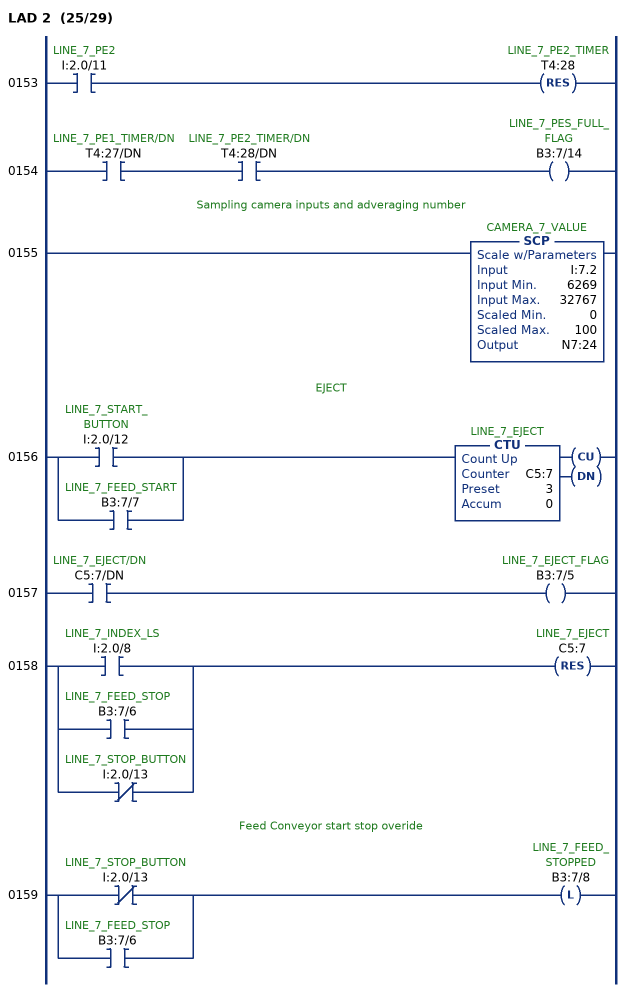
% Rung: 153 %  % edit flag set %
SOR XIC I:2.0/11 RES T4:28 EOR
%   I:2.0/11  LINE_7_PE2 %
%   T4:28  LINE_7_PE2_TIMER %
% Rung: 154 %  % edit flag set %
SOR XIC T4:27/DN XIC T4:28/DN OTE B3:7/14 EOR
%   T4:27  LINE_7_PE1_TIMER %
%   T4:28  LINE_7_PE2_TIMER %
%   B3:7/14  LINE_7_PES_FULL_FLAG %
% Rung: 155 %  % edit flag set %
% Sampling camera inputs and adveraging number %
SOR SCP I:7.2 6269 32767 0 100 N7:24 EOR
%   N7:24  CAMERA_7_VALUE %
% Rung: 156 %  % edit flag set %
% EJECT %
SOR BST XIC I:2.0/12 NXB XIC B3:7/7 BND CTU C5:7 3 0 EOR
%   I:2.0/12  LINE_7_START_BUTTON %
%   B3:7/7  LINE_7_FEED_START %
%   C5:7  LINE_7_EJECT %
% Rung: 157 %  % edit flag set %
SOR XIC C5:7/DN OTE B3:7/5 EOR
%   C5:7  LINE_7_EJECT %
%   B3:7/5  LINE_7_EJECT_FLAG %
% Rung: 158 %  % edit flag set %
SOR BST XIC I:2.0/8 NXB BST XIC B3:7/6 NXB XIO I:2.0/13 BND BND RES C5:7 EOR
%   I:2.0/8  LINE_7_INDEX_LS %
%   B3:7/6  LINE_7_FEED_STOP %
%   I:2.0/13  LINE_7_STOP_BUTTON %
%   C5:7  LINE_7_EJECT %
% Rung: 159 %  % edit flag set %
% Feed Conveyor start stop overide %
SOR BST XIO I:2.0/13 NXB XIC B3:7/6 BND OTL B3:7/8 EOR
%   I:2.0/13  LINE_7_STOP_BUTTON %
%   B3:7/6  LINE_7_FEED_STOP %
%   B3:7/8  LINE_7_FEED_STOPPED %

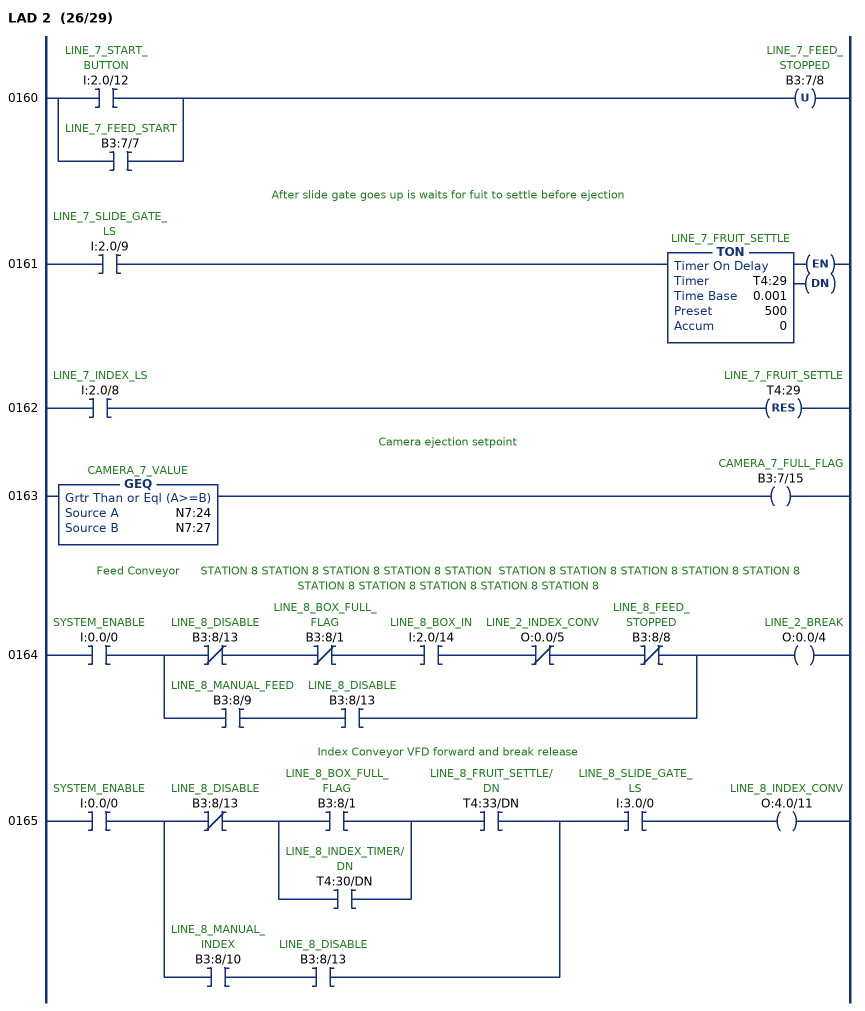
% Rung: 160 %  % edit flag set %
SOR BST XIC I:2.0/12 NXB XIC B3:7/7 BND OTU B3:7/8 EOR
%   I:2.0/12  LINE_7_START_BUTTON %
%   B3:7/7  LINE_7_FEED_START %
%   B3:7/8  LINE_7_FEED_STOPPED %
% Rung: 161 %  % edit flag set %
% After slide gate goes up is waits for fuit to settle before ejection %
SOR XIC I:2.0/9 TON T4:29 0.001 500 0 EOR
%   I:2.0/9  LINE_7_SLIDE_GATE_LS %
%   T4:29  LINE_7_FRUIT_SETTLE %
% Rung: 162 %  % edit flag set %
SOR XIC I:2.0/8 RES T4:29 EOR
%   I:2.0/8  LINE_7_INDEX_LS %
%   T4:29  LINE_7_FRUIT_SETTLE %
% Rung: 163 %  % edit flag set %
% Camera ejection setpoint %
SOR GEQ N7:24 N7:27 OTE B3:7/15 EOR
%   N7:24  CAMERA_7_VALUE %
%   N7:27  CAMERA_7_EJECT %
%   B3:7/15  CAMERA_7_FULL_FLAG %
% Rung: 164 %  % edit flag set %
% Feed Conveyor      STATION 8 STATION 8 STATION 8 STATION 8 STATION  STATION 8 STATION 8 STATION 8 STATION 8 STATION 8 STATION 8 STATION 8 STATION 8 STATION 8 STATION 8 %
SOR XIC I:0.0/0 BST XIO B3:8/13 XIO B3:8/1 XIC I:2.0/14 XIO O:0.0/5 XIO B3:8/8 NXB XIC B3:8/9 XIC B3:8/13 BND OTE O:0.0/4 EOR
%   I:0.0/0  SYSTEM_ENABLE %
%   B3:8/13  LINE_8_DISABLE %
%   B3:8/1  LINE_8_BOX_FULL_FLAG %
%   I:2.0/14  LINE_8_BOX_IN %
%   O:0.0/5  LINE_2_INDEX_CONV %
%   B3:8/8  LINE_8_FEED_STOPPED %
%   B3:8/9  LINE_8_MANUAL_FEED %
%   O:0.0/4  LINE_2_BREAK %
% Rung: 165 %  % edit flag set %
% Index Conveyor VFD forward and break release %
SOR XIC I:0.0/0 BST XIO B3:8/13 BST XIC B3:8/1 NXB XIC T4:30/DN BND XIC T4:33/DN NXB XIC B3:8/10 XIC B3:8/13 BND XIC I:3.0/0 OTE O:4.0/11 EOR
%   I:0.0/0  SYSTEM_ENABLE %
%   B3:8/13  LINE_8_DISABLE %
%   B3:8/1  LINE_8_BOX_FULL_FLAG %
%   T4:30  LINE_8_INDEX_TIMER %
%   T4:33  LINE_8_FRUIT_SETTLE %
%   B3:8/10  LINE_8_MANUAL_INDEX %
%   I:3.0/0  LINE_8_SLIDE_GATE_LS %
%   O:4.0/11  LINE_8_INDEX_CONV %

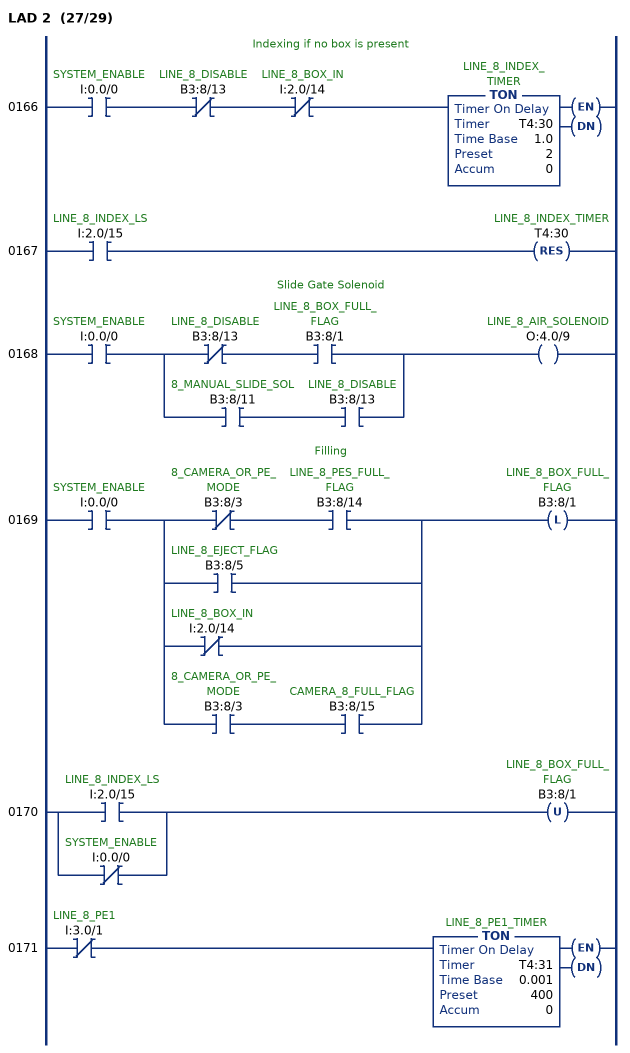
% Rung: 166 %  % edit flag set %
% Indexing if no box is present %
SOR XIC I:0.0/0 XIO B3:8/13 XIO I:2.0/14 TON T4:30 1.0 2 0 EOR
%   I:0.0/0  SYSTEM_ENABLE %
%   B3:8/13  LINE_8_DISABLE %
%   I:2.0/14  LINE_8_BOX_IN %
%   T4:30  LINE_8_INDEX_TIMER %
% Rung: 167 %  % edit flag set %
SOR XIC I:2.0/15 RES T4:30 EOR
%   I:2.0/15  LINE_8_INDEX_LS %
%   T4:30  LINE_8_INDEX_TIMER %
% Rung: 168 %  % edit flag set %
% Slide Gate Solenoid %
SOR XIC I:0.0/0 BST XIO B3:8/13 XIC B3:8/1 NXB XIC B3:8/11 XIC B3:8/13 BND OTE O:4.0/9 EOR
%   I:0.0/0  SYSTEM_ENABLE %
%   B3:8/13  LINE_8_DISABLE %
%   B3:8/1  LINE_8_BOX_FULL_FLAG %
%   B3:8/11  8_MANUAL_SLIDE_SOL %
%   O:4.0/9  LINE_8_AIR_SOLENOID %
% Rung: 169 %  % edit flag set %
% Filling %
SOR XIC I:0.0/0 BST XIO B3:8/3 XIC B3:8/14 NXB BST XIC B3:8/5 NXB BST XIO I:2.0/14 NXB XIC B3:8/3 XIC B3:8/15 BND BND BND OTL B3:8/1 EOR
%   I:0.0/0  SYSTEM_ENABLE %
%   B3:8/3  8_CAMERA_OR_PE_MODE %
%   B3:8/14  LINE_8_PES_FULL_FLAG %
%   B3:8/5  LINE_8_EJECT_FLAG %
%   I:2.0/14  LINE_8_BOX_IN %
%   B3:8/15  CAMERA_8_FULL_FLAG %
%   B3:8/1  LINE_8_BOX_FULL_FLAG %
% Rung: 170 %  % edit flag set %
SOR BST XIC I:2.0/15 NXB XIO I:0.0/0 BND OTU B3:8/1 EOR
%   I:2.0/15  LINE_8_INDEX_LS %
%   I:0.0/0  SYSTEM_ENABLE %
%   B3:8/1  LINE_8_BOX_FULL_FLAG %
% Rung: 171 %  % edit flag set %
SOR XIO I:3.0/1 TON T4:31 0.001 400 0 EOR
%   I:3.0/1  LINE_8_PE1 %
%   T4:31  LINE_8_PE1_TIMER %

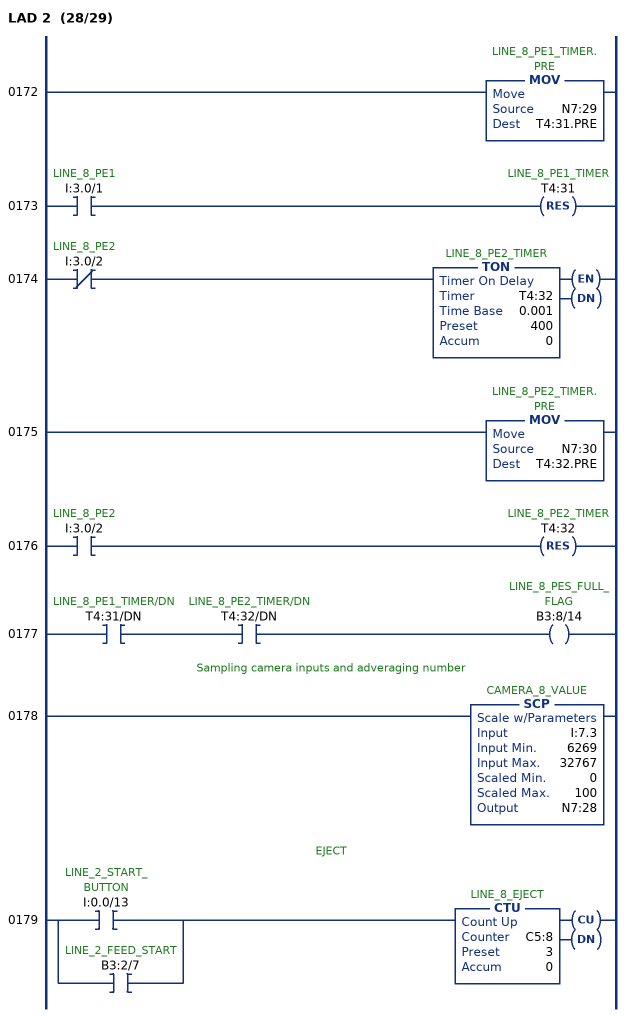
% Rung: 172 %  % edit flag set %
SOR MOV N7:29 T4:31.PRE EOR
%   N7:29  LINE_8_PE1_TIME_MOV %
%   T4:31  LINE_8_PE1_TIMER %
% Rung: 173 %  % edit flag set %
SOR XIC I:3.0/1 RES T4:31 EOR
%   I:3.0/1  LINE_8_PE1 %
%   T4:31  LINE_8_PE1_TIMER %
% Rung: 174 %  % edit flag set %
SOR XIO I:3.0/2 TON T4:32 0.001 400 0 EOR
%   I:3.0/2  LINE_8_PE2 %
%   T4:32  LINE_8_PE2_TIMER %
% Rung: 175 %  % edit flag set %
SOR MOV N7:30 T4:32.PRE EOR
%   N7:30  LINE_8_PE2_TIME_MOV %
%   T4:32  LINE_8_PE2_TIMER %
% Rung: 176 %  % edit flag set %
SOR XIC I:3.0/2 RES T4:32 EOR
%   I:3.0/2  LINE_8_PE2 %
%   T4:32  LINE_8_PE2_TIMER %
% Rung: 177 %  % edit flag set %
SOR XIC T4:31/DN XIC T4:32/DN OTE B3:8/14 EOR
%   T4:31  LINE_8_PE1_TIMER %
%   T4:32  LINE_8_PE2_TIMER %
%   B3:8/14  LINE_8_PES_FULL_FLAG %
% Rung: 178 %  % edit flag set %
% Sampling camera inputs and adveraging number %
SOR SCP I:7.3 6269 32767 0 100 N7:28 EOR
%   N7:28  CAMERA_8_VALUE %
% Rung: 179 %  % edit flag set %
% EJECT %
SOR BST XIC I:0.0/13 NXB XIC B3:2/7 BND CTU C5:8 3 0 EOR
%   I:0.0/13  LINE_2_START_BUTTON %
%   B3:2/7  LINE_2_FEED_START %
%   C5:8  LINE_8_EJECT %

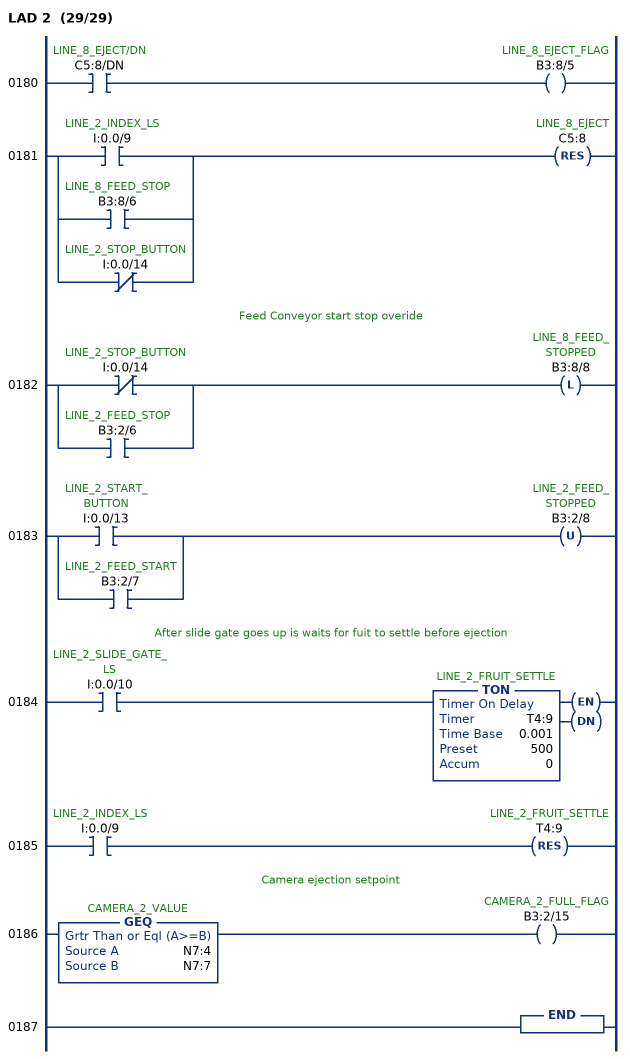
% Rung: 180 %  % edit flag set %
SOR XIC C5:8/DN OTE B3:8/5 EOR
%   C5:8  LINE_8_EJECT %
%   B3:8/5  LINE_8_EJECT_FLAG %
% Rung: 181 %  % edit flag set %
SOR BST XIC I:0.0/9 NXB BST XIC B3:8/6 NXB XIO I:0.0/14 BND BND RES C5:8 EOR
%   I:0.0/9  LINE_2_INDEX_LS %
%   B3:8/6  LINE_8_FEED_STOP %
%   I:0.0/14  LINE_2_STOP_BUTTON %
%   C5:8  LINE_8_EJECT %
% Rung: 182 %  % edit flag set %
% Feed Conveyor start stop overide %
SOR BST XIO I:0.0/14 NXB XIC B3:2/6 BND OTL B3:8/8 EOR
%   I:0.0/14  LINE_2_STOP_BUTTON %
%   B3:2/6  LINE_2_FEED_STOP %
%   B3:8/8  LINE_8_FEED_STOPPED %
% Rung: 183 %  % edit flag set %
SOR BST XIC I:0.0/13 NXB XIC B3:2/7 BND OTU B3:2/8 EOR
%   I:0.0/13  LINE_2_START_BUTTON %
%   B3:2/7  LINE_2_FEED_START %
%   B3:2/8  LINE_2_FEED_STOPPED %
% Rung: 184 %  % edit flag set %
% After slide gate goes up is waits for fuit to settle before ejection %
SOR XIC I:0.0/10 TON T4:9 0.001 500 0 EOR
%   I:0.0/10  LINE_2_SLIDE_GATE_LS %
%   T4:9  LINE_2_FRUIT_SETTLE %
% Rung: 185 %  % edit flag set %
SOR XIC I:0.0/9 RES T4:9 EOR
%   I:0.0/9  LINE_2_INDEX_LS %
%   T4:9  LINE_2_FRUIT_SETTLE %
% Rung: 186 %  % edit flag set %
% Camera ejection setpoint %
SOR GEQ N7:4 N7:7 OTE B3:2/15 EOR
%   N7:4  CAMERA_2_VALUE %
%   N7:7  LINE_2_CAMERA_EJECT %
%   B3:2/15  CAMERA_2_FULL_FLAG %
% Rung: 187 %
SOR END EOR

OTHER DOCUMENTED ADDRESSES
  B3:0/4  1_BOX_FULL_UNLATCH  "Box Full Unlatch"
  B3:2/4  2_BOX_FULL_UNLATCH
  B3:3/4  3_BOX_FULL_UNLATCH
  B3:4/4  4_BOX_FULL_UNLATCH
  B3:5/4  5_BOX_FULL_UNLATCH
  B3:6/4  6_BOX_FULL_UNLATCH
  B3:7/4  7_BOX_FULL_UNLATCH
  B3:8/4  8_BOX_FULL_UNLATCH
  B3:8/7  LINE_8_FEED_START
  C5:0.ACC  "Counter"
  C5:0/DN  COUNT_DONE
  I:3.0/3  LINE_8_START_BUTTON
  I:3.0/4  LINE_8_STOP_BUTTON
  I:6.0/0  CAMERA_1  "Camera 1 4-20 input"
  I:7.0/0  CAMERA_5  "Camera 1 4-20 input"
  N7:31  CAMERA_8_EJECT
  O:4.0/10  LINE_8_BREAK

REVISION NOTES
  0: Simplified

DATA TABLE (non-zero values as saved)
DATA B3
% B3:0 % 0X0004 0X000B 0X0000 0X0000 0X0000 0X0000 0X0000 0X0000 0X0000 0X0001
DATA T4
% .PRE .ACC %
% T4:0 % 2 0
% T4:1 % 400 0
% T4:2 % 1 1
% T4:3 % 1 0
% T4:4 % 400 0
% T4:5 % 500 0
% T4:6 % 1440 1530
DATA C5
% .PRE .ACC %
% C5:0 % 6 1
% C5:1 % 3 0
DATA N7
% N7:0 % 36 51 51 51 51 52 102 153 204 256
% N7:10 % 51 1470 400 400 50 0 0 0 0 0
DATA F8
% F8:0 % 0 22161 86.55965
